FUNCTION_BLOCK FB_FRAMESELECTOR
VAR
	//SelectedFrame	: FrameSelect;
	SelectedFrame : INT := 0;
	ShowFrame		: BOOL;
END_VAR

END_FUNCTION_BLOCK

(* stored: Version 1.1.0.1, ProductVersion 3.1.4024.15
   POU FB_FRAMESELECTOR: Id {a913e27a-a3ee-4710-8068-da1f861e577a}, SpecialFunc None *)
